{attribute 'qualified_only'}
VAR_GLOBAL PERSISTENT
	Tags: AdsTagsExtraAlarms;
END_VAR

(* stored: Version 1.1.0.1, ProductVersion 3.1.4024.6
   GVL ADS_ExtraAlarms: Id {b8fbe193-c8ef-4590-92ae-2729a01f5fcc} *)
